// TIA Portal V20 export
DATA_BLOCK "DB_DigitalInputsBW_Station"   // DB2214
// stored: AutoNumber false, InstanceOfName FB_DigitalInputsBW_Station, InstanceOfType FB
"FB_DigitalInputsBW_Station"
   // VAR
   //    sUndrilledPartCtrl { S7_SetPoint := 'True'} : "FB_DigitalInput";
   //    sDrilledPartCtrl { S7_SetPoint := 'True'} : "FB_DigitalInput";
   //    sBwCtrl { S7_SetPoint := 'True'} : "FB_DigitalInput";
   // END_VAR
BEGIN
END_DATA_BLOCK
